// SIMATIC S7-200 project (STEP 7-Micro/WIN), CPU 221 REL 01.10

SYMBOL_TABLE USER1
reached_down     Q0.3     // Chegou ao sensor de baixo (P0.3)
reached_left     Q0.5     // Chegou ao sensor da esquerda (P0.5)
go_down          Q2.3
reached_up       Q0.4     // Chegou ao sensor de cima (P0.4)
go_left          Q2.1
go_up            Q2.2
reached_right    Q0.6     // Chegou ao sensor da direita (P0.6)
simple_wash_selected I2.0
SIMPLE_WASH      M0.0
go_right         Q2.0
complete_wash_selected I2.1
power_down_selected I2.3
stop_selected    I2.4
resume_selected  I2.5
escovas_horizontais Q2.5     // Activar escovas horizontais
escovas_verticais Q2.4     // Activar escovas verticais
left_infra_red   Q0.1
right_infra_red  Q0.2
COMPLETE_WASH    M0.1
POWER_DOWN       M0.2
STOP_SYSTEM      M0.3
RESUME_SYSTEM    M0.4
END_SYMBOL_TABLE

ORGANIZATION_BLOCK Program_Block:OB1
TITLE=PROGRAM COMMENTS
BEGIN
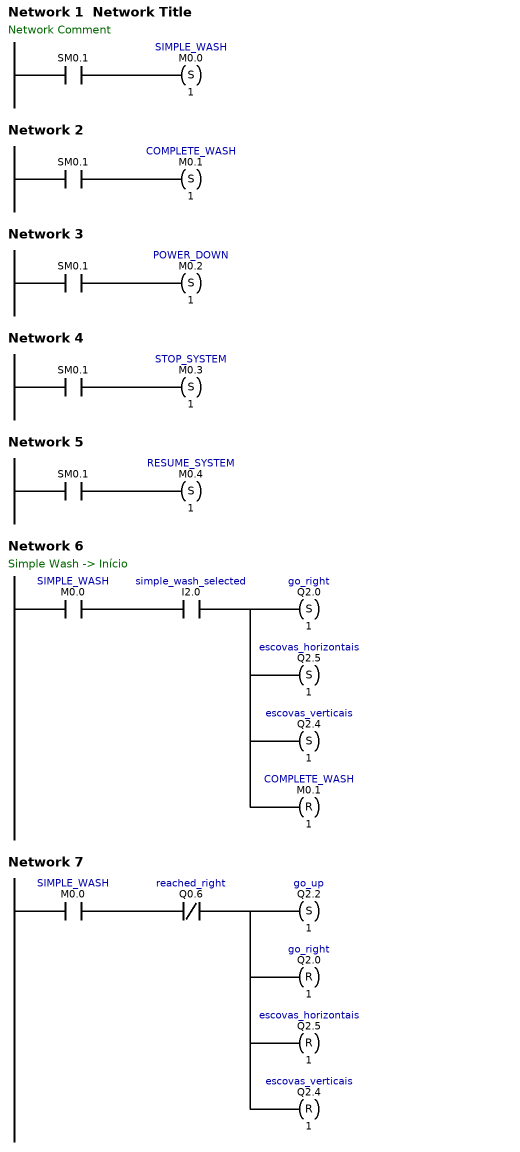
Network 1 // Network Title
// Network Comment
LD     SM0.1
S      SIMPLE_WASH:M0.0, 1
Network 2
LD     SM0.1
S      COMPLETE_WASH:M0.1, 1
Network 3
LD     SM0.1
S      POWER_DOWN:M0.2, 1
Network 4
LD     SM0.1
S      STOP_SYSTEM:M0.3, 1
Network 5
LD     SM0.1
S      RESUME_SYSTEM:M0.4, 1
Network 6
// Simple Wash -> Início
LD     SIMPLE_WASH:M0.0
A      simple_wash_selected:I2.0
S      go_right:Q2.0, 1
S      escovas_horizontais:Q2.5, 1
S      escovas_verticais:Q2.4, 1
R      COMPLETE_WASH:M0.1, 1
Network 7
LD     SIMPLE_WASH:M0.0
AN     reached_right:Q0.6
S      go_up:Q2.2, 1
R      go_right:Q2.0, 1
R      escovas_horizontais:Q2.5, 1
R      escovas_verticais:Q2.4, 1
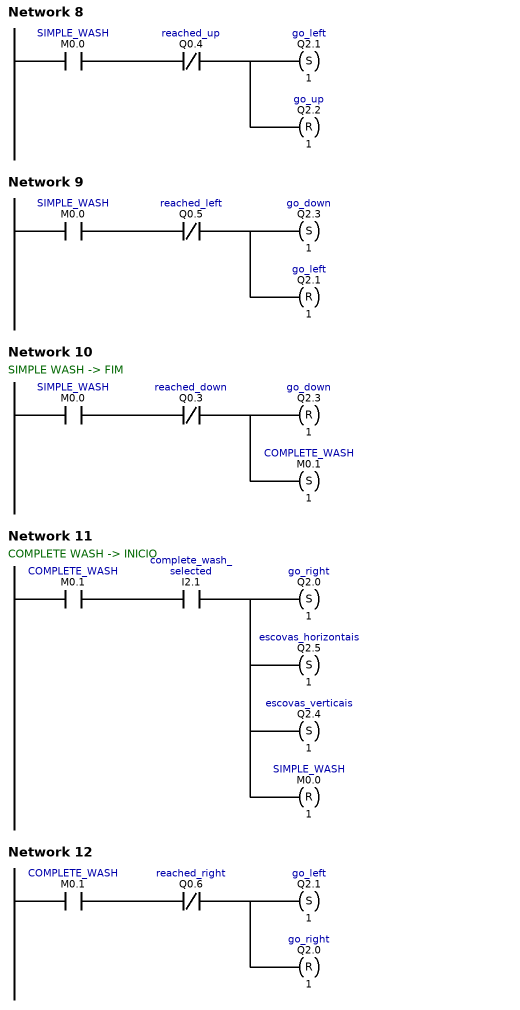
Network 8
LD     SIMPLE_WASH:M0.0
AN     reached_up:Q0.4
S      go_left:Q2.1, 1
R      go_up:Q2.2, 1
Network 9
LD     SIMPLE_WASH:M0.0
AN     reached_left:Q0.5
S      go_down:Q2.3, 1
R      go_left:Q2.1, 1
Network 10
// SIMPLE WASH -> FIM
LD     SIMPLE_WASH:M0.0
AN     reached_down:Q0.3
R      go_down:Q2.3, 1
S      COMPLETE_WASH:M0.1, 1
Network 11
// COMPLETE WASH -> INICIO
LD     COMPLETE_WASH:M0.1
A      complete_wash_selected:I2.1
S      go_right:Q2.0, 1
S      escovas_horizontais:Q2.5, 1
S      escovas_verticais:Q2.4, 1
R      SIMPLE_WASH:M0.0, 1
Network 12
LD     COMPLETE_WASH:M0.1
AN     reached_right:Q0.6
S      go_left:Q2.1, 1
R      go_right:Q2.0, 1
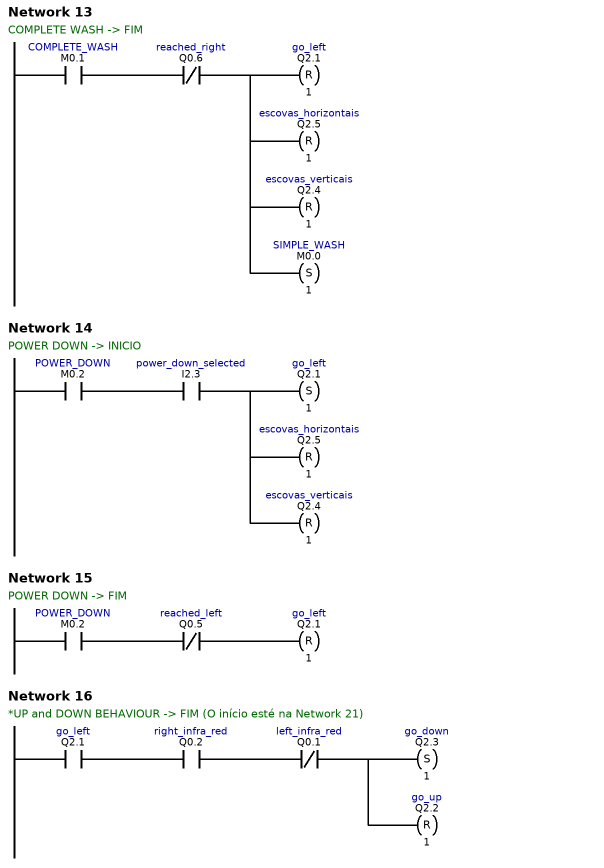
Network 13
// COMPLETE WASH -> FIM
LD     COMPLETE_WASH:M0.1
AN     reached_right:Q0.6
R      go_left:Q2.1, 1
R      escovas_horizontais:Q2.5, 1
R      escovas_verticais:Q2.4, 1
S      SIMPLE_WASH:M0.0, 1
Network 14
// POWER DOWN -> INICIO
LD     POWER_DOWN:M0.2
A      power_down_selected:I2.3
S      go_left:Q2.1, 1
R      escovas_horizontais:Q2.5, 1
R      escovas_verticais:Q2.4, 1
Network 15
// POWER DOWN -> FIM
LD     POWER_DOWN:M0.2
AN     reached_left:Q0.5
R      go_left:Q2.1, 1
Network 16
// *UP and DOWN BEHAVIOUR -> FIM (O início esté na Network 21)
LD     go_left:Q2.1
A      right_infra_red:Q0.2
AN     left_infra_red:Q0.1
S      go_down:Q2.3, 1
R      go_up:Q2.2, 1
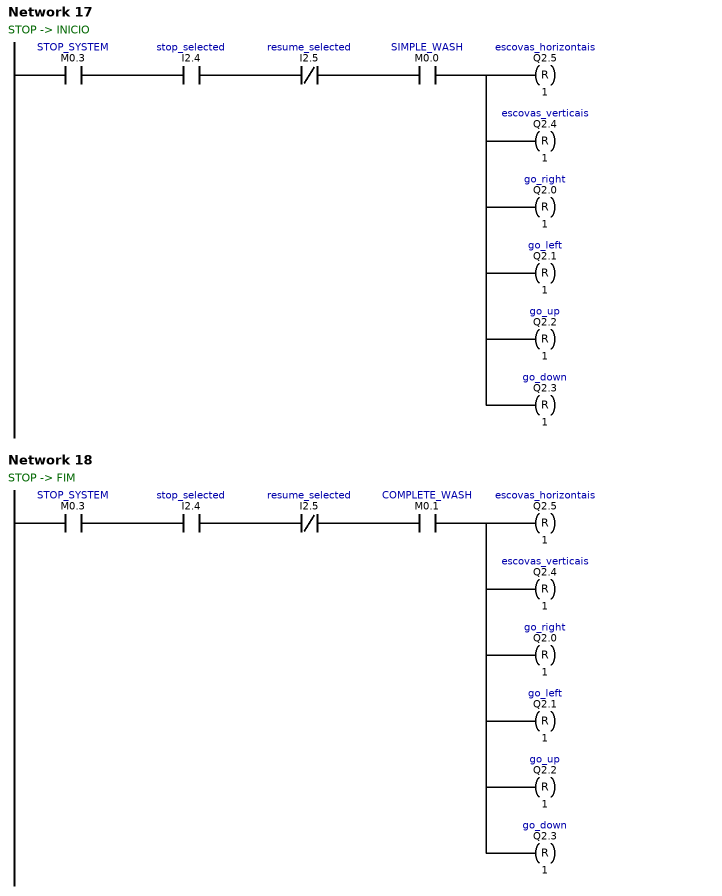
Network 17
// STOP -> INICIO
LD     STOP_SYSTEM:M0.3
A      stop_selected:I2.4
AN     resume_selected:I2.5
A      SIMPLE_WASH:M0.0
R      escovas_horizontais:Q2.5, 1
R      escovas_verticais:Q2.4, 1
R      go_right:Q2.0, 1
R      go_left:Q2.1, 1
R      go_up:Q2.2, 1
R      go_down:Q2.3, 1
Network 18
// STOP -> FIM
LD     STOP_SYSTEM:M0.3
A      stop_selected:I2.4
AN     resume_selected:I2.5
A      COMPLETE_WASH:M0.1
R      escovas_horizontais:Q2.5, 1
R      escovas_verticais:Q2.4, 1
R      go_right:Q2.0, 1
R      go_left:Q2.1, 1
R      go_up:Q2.2, 1
R      go_down:Q2.3, 1
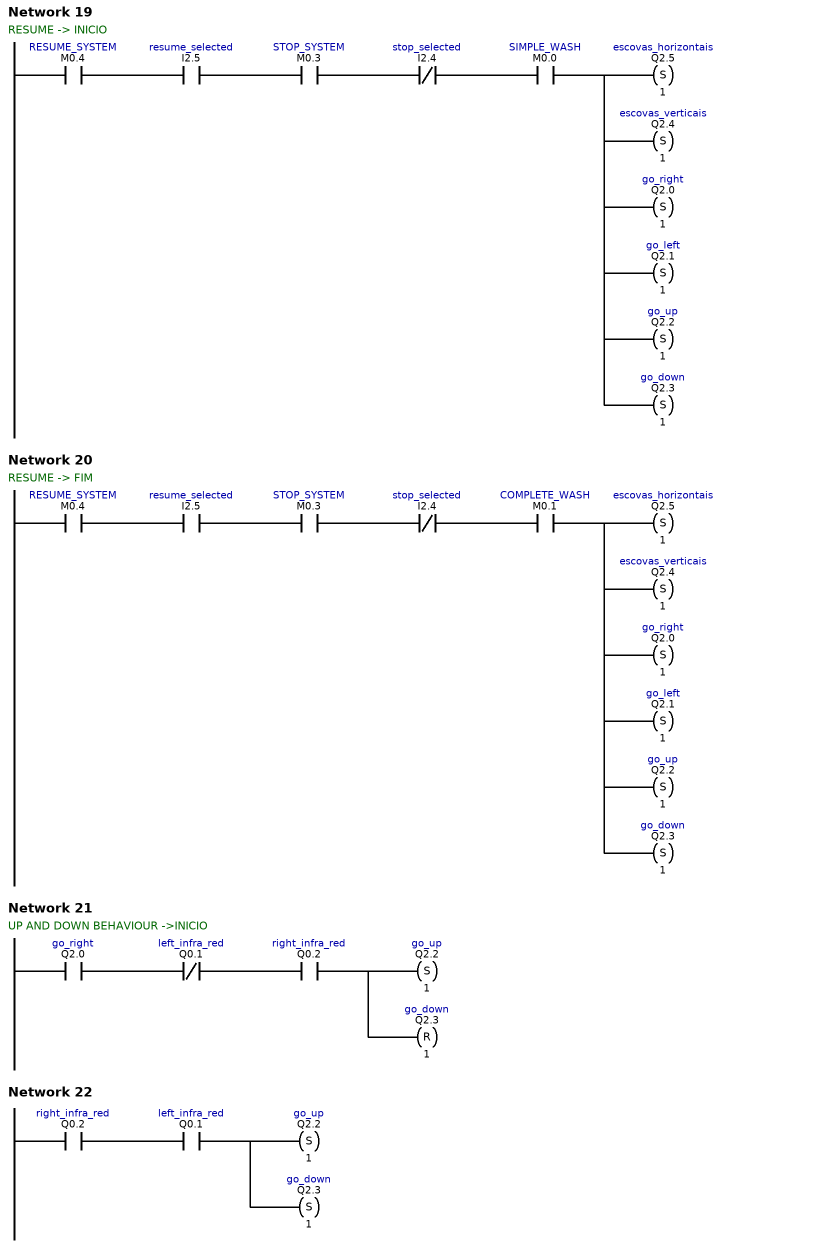
Network 19
// RESUME -> INICIO
LD     RESUME_SYSTEM:M0.4
A      resume_selected:I2.5
A      STOP_SYSTEM:M0.3
AN     stop_selected:I2.4
A      SIMPLE_WASH:M0.0
S      escovas_horizontais:Q2.5, 1
S      escovas_verticais:Q2.4, 1
S      go_right:Q2.0, 1
S      go_left:Q2.1, 1
S      go_up:Q2.2, 1
S      go_down:Q2.3, 1
Network 20
// RESUME -> FIM
LD     RESUME_SYSTEM:M0.4
A      resume_selected:I2.5
A      STOP_SYSTEM:M0.3
AN     stop_selected:I2.4
A      COMPLETE_WASH:M0.1
S      escovas_horizontais:Q2.5, 1
S      escovas_verticais:Q2.4, 1
S      go_right:Q2.0, 1
S      go_left:Q2.1, 1
S      go_up:Q2.2, 1
S      go_down:Q2.3, 1
Network 21
// UP AND DOWN BEHAVIOUR ->INICIO
LD     go_right:Q2.0
AN     left_infra_red:Q0.1
A      right_infra_red:Q0.2
S      go_up:Q2.2, 1
R      go_down:Q2.3, 1
Network 22
LD     right_infra_red:Q0.2
A      left_infra_red:Q0.1
S      go_up:Q2.2, 1
S      go_down:Q2.3, 1
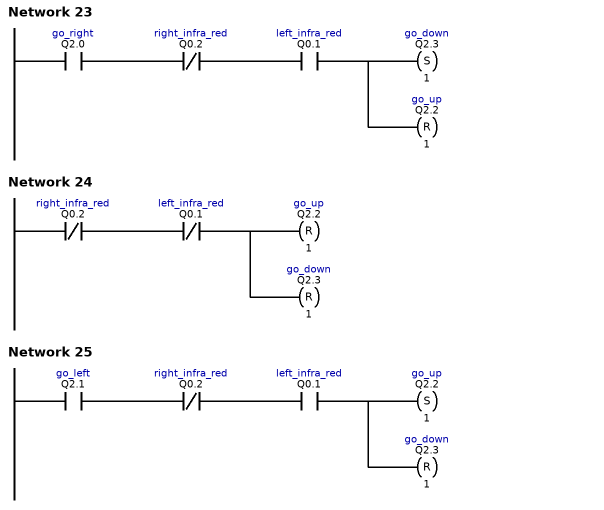
Network 23
LD     go_right:Q2.0
AN     right_infra_red:Q0.2
A      left_infra_red:Q0.1
S      go_down:Q2.3, 1
R      go_up:Q2.2, 1
Network 24
LDN    right_infra_red:Q0.2
AN     left_infra_red:Q0.1
R      go_up:Q2.2, 1
R      go_down:Q2.3, 1
Network 25
LD     go_left:Q2.1
AN     right_infra_red:Q0.2
A      left_infra_red:Q0.1
S      go_up:Q2.2, 1
R      go_down:Q2.3, 1
END_ORGANIZATION_BLOCK
